{attribute 'GeneratedUsingTerminal: KL9260'}
{attribute addProperty BoxType "KL9260"}
{attribute addProperty Description ""}
{attribute addProperty Physics ""}
{attribute addProperty Id "Channel_1AT %I*Channel_64AAC8C70"}
{attribute addProperty CRC "2347652594"}
{attribute addProperty Size "0"}
TYPE KL9260_8BEE55F2 :
STRUCT
	{attribute addProperty Name "Channel_1"}
	Channel_1 : Channel_64AAC8C7;
END_STRUCT
END_TYPE

(* stored: Version 1.2.0.0, ProductVersion 3.1.4024.9
   DUT KL9260_8BEE55F2: Id {0fb9b2df-9d6e-439b-a0f2-d61e9c76a45c} *)
